FUNCTION_BLOCK FB_3eTI_iMesh_Base
VAR_INPUT
	
	// THIS IS FOR THE ISA100.11A GATEWAY
	mbAddrs : ARRAY[0..3] OF MODBUS_DATA_MAP :=  [ 
			(_ipAddress := '192.168.254.253', _startAddress:= 6), 
			(_ipAddress := '192.168.254.253', _startAddress:= 18),
			(_ipAddress := '192.168.254.253', _startAddress:= 30),
			(_ipAddress := '192.168.254.253', _startAddress:= 42)
		];
		
END_VAR

VAR
	fbReadMB 	: FB_ReadModbus;
	ii			: INT:=0;
END_VAR

VAR_OUTPUT
END_VAR

VAR
END_VAR

//
// BEGIN PRODUCE THE DATA
//
// XMEAS values will come from the external TESIM program using ADS

// VOLTAGES
XMEAS_IO_VOUT[XMEAS_IO_IDX.A_FLOW]		:= pv_float_to_dac(pv:=XMEAS[XMEAS_IDX.A_FLOW],		pv_max:=G_PARAMS.A_FLOW_MAX, pv_min:=G_PARAMS.A_FLOW_MIN, dac_max:=VOUT_WD_MAX, dac_min:=0);
XMEAS_IO_VOUT[XMEAS_IO_IDX.D_FLOW]		:= pv_float_to_dac(pv:=XMEAS[XMEAS_IDX.D_FLOW],		pv_max:=G_PARAMS.D_FLOW_MAX, pv_min:=G_PARAMS.D_FLOW_MIN, dac_max:=VOUT_WD_MAX, dac_min:=0);
XMEAS_IO_VOUT[XMEAS_IO_IDX.E_FLOW]		:= pv_float_to_dac(pv:=XMEAS[XMEAS_IDX.E_FLOW],		pv_max:=G_PARAMS.E_FLOW_MAX, pv_min:=G_PARAMS.E_FLOW_MIN, dac_max:=VOUT_WD_MAX, dac_min:=0);
XMEAS_IO_VOUT[XMEAS_IO_IDX.AC_FLOW]	:= pv_float_to_dac(pv:=XMEAS[XMEAS_IDX.AC_FLOW],	pv_max:=G_PARAMS.AC_FLOW_MAX, pv_min:=G_PARAMS.AC_FLOW_MIN, dac_max:=VOUT_WD_MAX, dac_min:=0);

//
// BEGIN MODBUS POLLING SEGMENT from the GATEWAY
//
fbReadMB(addrs := mbAddrs );

// poll modbus registers
G_IO.MBS_XMEAS_RAW[XMEAS_MBS_IDX.A_FLOW] := fbReadMB.registerValues[XMEAS_MBS_IDX.A_FLOW] + MBS_XMEAS_CAL_OFFSET[1];
G_IO.MBS_XMEAS_RAW[XMEAS_MBS_IDX.D_FLOW] := fbReadMB.registerValues[XMEAS_MBS_IDX.D_FLOW]+ MBS_XMEAS_CAL_OFFSET[2];
G_IO.MBS_XMEAS_RAW[XMEAS_MBS_IDX.E_FLOW] := fbReadMB.registerValues[XMEAS_MBS_IDX.E_FLOW] + MBS_XMEAS_CAL_OFFSET[3];
G_IO.MBS_XMEAS_RAW[XMEAS_MBS_IDX.AC_FLOW] := fbReadMB.registerValues[XMEAS_MBS_IDX.AC_FLOW] + MBS_XMEAS_CAL_OFFSET[4];

// convert raw modbus signals to process signals
G_IO.MBS_XMEAS[XMEAS_MBS_IDX.A_FLOW]	:=	LREAL_TO_REAL(adc_to_float_pv(G_IO.MBS_XMEAS_RAW[XMEAS_MBS_IDX.A_FLOW],		pv_max:=G_PARAMS.A_FLOW_MAX, 		pv_min:=G_PARAMS.A_FLOW_MIN, 	i_max:=G_PARAMS.VOUT_MAX, i_min:=G_PARAMS.VOUT_MIN));
G_IO.MBS_XMEAS[XMEAS_MBS_IDX.D_FLOW]	:=	LREAL_TO_REAL(adc_to_float_pv(G_IO.MBS_XMEAS_RAW[XMEAS_MBS_IDX.D_FLOW],		pv_max:=G_PARAMS.D_FLOW_MAX, 		pv_min:=G_PARAMS.D_FLOW_MIN, 	i_max:=G_PARAMS.VOUT_MAX, i_min:=G_PARAMS.VOUT_MIN));
G_IO.MBS_XMEAS[XMEAS_MBS_IDX.E_FLOW]	:=	LREAL_TO_REAL(adc_to_float_pv(G_IO.MBS_XMEAS_RAW[XMEAS_MBS_IDX.E_FLOW],		pv_max:=G_PARAMS.E_FLOW_MAX, 		pv_min:=G_PARAMS.E_FLOW_MIN, 	i_max:=G_PARAMS.VOUT_MAX, i_min:=G_PARAMS.VOUT_MIN));
G_IO.MBS_XMEAS[XMEAS_MBS_IDX.AC_FLOW]	:=	LREAL_TO_REAL(adc_to_float_pv(G_IO.MBS_XMEAS_RAW[XMEAS_MBS_IDX.AC_FLOW],	pv_max:=G_PARAMS.AC_FLOW_MAX, 	pv_min:=G_PARAMS.AC_FLOW_MIN, i_max:=G_PARAMS.VOUT_MAX, i_min:=G_PARAMS.VOUT_MIN));

// capture the received state of XMEAS
FOR ii := 1 TO 41 DO
	XMEAS_RX[ii]:=XMEAS[ii];
END_FOR
XMEAS_RX[XMEAS_IDX.A_FLOW] := G_IO.MBS_XMEAS[XMEAS_MBS_IDX.A_FLOW];
XMEAS_RX[XMEAS_IDX.D_FLOW] := G_IO.MBS_XMEAS[XMEAS_MBS_IDX.D_FLOW];
XMEAS_RX[XMEAS_IDX.E_FLOW] := G_IO.MBS_XMEAS[XMEAS_MBS_IDX.E_FLOW];
XMEAS_RX[XMEAS_IDX.AC_FLOW] := G_IO.MBS_XMEAS[XMEAS_MBS_IDX.AC_FLOW];


//
// END MODBUS POLLING SEGMENT from the GATEWAY
//

END_FUNCTION_BLOCK

(* stored: Version 1.1.0.1, ProductVersion 3.1.0.36
   POU FB_3eTI_iMesh_Base: Id {c24ff66a-4461-44bb-a3fd-0d65c26a2169}, SpecialFunc None *)
